// TIA Portal project "hassn_and_musa" (V17)
// Vorlageprojekt für das Buch mit Zielsystem S7-1200

(* hardware
DEVICE "S7-1200-Station_1"  S7-1200 Station
   slot 0: "Baugruppenträger_0"  Rack  V1.0
   slot 1: "PLC_1"  CPU 1211C DC/DC/DC  6ES7 211-1AE40-0XB0  V4.1
DEVICE "HMI_1"  TP700 Comfort
   slot 0: "HMI_1"  TP700 Comfort  6AV2 124-0GC01-0AX0  15.0.0.0
   slot 1: "HMI_RT_1"  TP700 Comfort  6AV2 124-0GC01-0AX0  15.0.0.0
   slot 5: "HMI_1.IE_CP_1"  PROFINET Interface  15.0.0.0
      slot 1: "PROFINET Interface_1"  PROFINET Interface
         slot 1: "Port_1"  Port
         slot 2: "Port_2"  Port
   slot 7: "HMI_1.MPI/DP_CP_1"  MPI/DP Interface  15.0.0.0
*)

// ===== PLC "PLC_1"  CPU 1211C DC/DC/DC =====

VAR_GLOBAL   // PLC tag table "Standard-Variablentabelle"
   "StartButton" AT %I0.0 : Bool;
   "StopButton" AT %I0.1 : Bool;
   "StartLight" AT %Q0.0 : Bool;
   "StopLIght" AT %Q0.1 : Bool;
   "emergency stop" AT %I0.2 : Bool;
   "FlipFlop1" AT %M0.0 : Bool;
   "FlipFlop2" AT %M0.1 : Bool;
   "First Conveyor" AT %Q0.4 : Bool;
   "Second Conveyor" AT %Q0.5 : Bool;
   "Vision Sensor" AT %ID34 : DInt;
   "Third Conveyor" AT %Q0.6 : Bool;
   "pusher" AT %Q0.3 : Bool;
   "pusherbacklimit" AT %I0.3 : Bool;
   "pusherfrontlimit" AT %I0.4 : Bool;
   "SensorForblue" AT %I0.5 : Bool;
   "SensorForGreen" AT %I0.6 : Bool;
   "MoveZBlue" AT %Q0.7 : Bool;
   "MoveZGreen" AT %Q1.0 : Bool;
   "Tag_1" AT %M0.2 : Bool;
   "Tag_2" AT %M0.3 : Bool;
   "Tag_3" AT %M0.4 : Bool;
   "Tag_4" AT %M0.5 : Bool;
   "SensorBlueCount" AT %I0.7 : Bool;
   "SensorGrCount" AT %I1.0 : Bool;
   "Tag_5" AT %M0.6 : Bool;
   "Tag_6" AT %M0.7 : Bool;
   "Tag_7" AT %M1.0 : Bool;
   "Tag_8" AT %M1.1 : Bool;
   "Tag_9" AT %M1.2 : Bool;
END_VAR

DATA_BLOCK "HMI"   // DB1
{ S7_Optimized_Access := 'TRUE' }
VERSION : 0.1
   VAR
      "blue boxes" : Int;
      "Reset Count" : Bool;
      "Green boxes" : Int;
      "emergency hmi" : Bool;
      start : Bool;
      stop : Bool;
   END_VAR
BEGIN
END_DATA_BLOCK

// folder: System blocks/Program resources

DATA_BLOCK "IEC_Counter_0_DB"   // DB2
{ S7_Optimized_Access := 'TRUE' }
AUTHOR : Simatic
FAMILY : IEC
NAME : CNTR
VERSION : 1.0
// stored: InstanceOfName IEC_COUNTER
"IEC_COUNTER"
BEGIN
END_DATA_BLOCK

DATA_BLOCK "IEC_Counter_0_DB_1"   // DB3
{ S7_Optimized_Access := 'TRUE' }
AUTHOR : Simatic
FAMILY : IEC
NAME : CNTR
VERSION : 1.0
// stored: InstanceOfName IEC_COUNTER
"IEC_COUNTER"
BEGIN
END_DATA_BLOCK

// folder: (top level)

FUNCTION "Buttonlights" : Void   // FC1, LAD
{ S7_Optimized_Access := 'TRUE' }
VERSION : 0.1
BEGIN

REGION Network 1
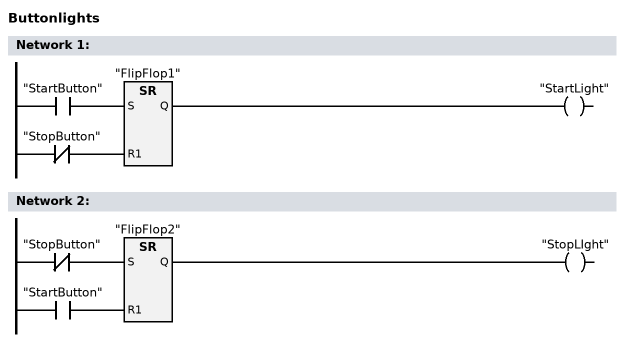
   RUNG wire#powerrail
      Contact( "StartButton" )
      S_SR(operand := "FlipFlop1", r1 := wire#w1)
      Coil( "StartLight" )
   END_RUNG
   RUNG wire#powerrail
      I_Contact( "StopButton" )
   END_RUNG wire#w1
   // the same network as SCL:
   IF "StartButton" THEN
       "FlipFlop1" := TRUE;   // SR flip-flop
   END_IF;
   IF NOT "StopButton" THEN "FlipFlop1" := FALSE; END_IF;
   "StartLight" := "FlipFlop1";
END_REGION

REGION Network 2
   RUNG wire#powerrail
      I_Contact( "StopButton" )
      S_SR(operand := "FlipFlop2", r1 := wire#w1)
      Coil( "StopLIght" )
   END_RUNG
   RUNG wire#powerrail
      Contact( "StartButton" )
   END_RUNG wire#w1
   // the same network as SCL:
   IF NOT "StopButton" THEN
       "FlipFlop2" := TRUE;   // SR flip-flop
   END_IF;
   IF "StartButton" THEN "FlipFlop2" := FALSE; END_IF;
   "StopLIght" := "FlipFlop2";
END_REGION
END_FUNCTION

FUNCTION "StartConvFromFactory" : Void   // FC2, LAD
{ S7_Optimized_Access := 'TRUE' }
VERSION : 0.1
BEGIN

REGION Network 1
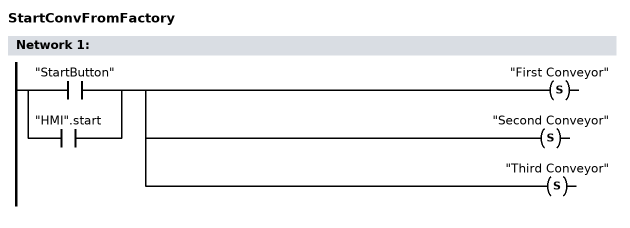
   RUNG wire#powerrail
      Contact( "StartButton" )
      wire#w1
      S_Coil( "First Conveyor" )
   END_RUNG
   RUNG wire#powerrail
      Contact( "HMI".start )
   END_RUNG wire#w1
   RUNG wire#w1
      S_Coil( "Second Conveyor" )
   END_RUNG
   RUNG wire#w1
      S_Coil( "Third Conveyor" )
   END_RUNG
   // the same network as SCL:
   IF "StartButton" OR "HMI".start THEN
       "First Conveyor" := TRUE;
       "Second Conveyor" := TRUE;
       "Third Conveyor" := TRUE;
   END_IF;
END_REGION
END_FUNCTION

FUNCTION "PushGreen" : Void   // FC3, SCL
{ S7_Optimized_Access := 'TRUE' }
VERSION : 0.1
BEGIN

   IF "Vision Sensor" = 4 AND "pusherbacklimit" = 1 THEN
       "pusher" := 1;
   ELSIF "Vision Sensor" <> 4 AND "pusherfrontlimit" = 1 THEN
       "pusher" := 0;
   END_IF;
END_FUNCTION

FUNCTION "Put the tags" : Void   // FC4, LAD
{ S7_Optimized_Access := 'TRUE' }
VERSION : 0.1
   VAR_TEMP   // added for the SCL form of the ladder/FBD networks
      _w1 : Bool;
      _w2 : Bool;
      _w3 : Bool;
      _w4 : Bool;
   END_VAR
BEGIN

REGION Network 1
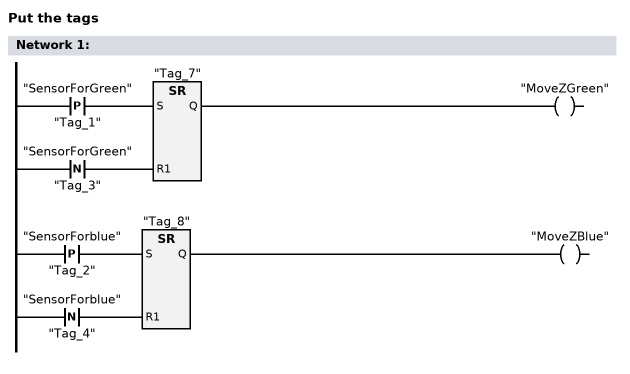
   RUNG wire#powerrail
      P_Contact(operand := "SensorForGreen", bit := "Tag_1")
      S_SR(operand := "Tag_7", r1 := wire#w1)
      Coil( "MoveZGreen" )
   END_RUNG
   RUNG wire#powerrail
      N_Contact(operand := "SensorForGreen", bit := "Tag_3")
   END_RUNG wire#w1
   RUNG wire#powerrail
      P_Contact(operand := "SensorForblue", bit := "Tag_2")
      S_SR(operand := "Tag_8", r1 := wire#w2)
      Coil( "MoveZBlue" )
   END_RUNG
   RUNG wire#powerrail
      N_Contact(operand := "SensorForblue", bit := "Tag_4")
   END_RUNG wire#w2
   // the same network as SCL:
   #_w1 := "SensorForGreen" AND NOT "Tag_1";   // rising edge of "SensorForGreen"
   "Tag_1" := "SensorForGreen";
   #_w2 := NOT "SensorForGreen" AND "Tag_3";   // falling edge of "SensorForGreen"
   "Tag_3" := "SensorForGreen";
   IF #_w1 THEN
       "Tag_7" := TRUE;   // SR flip-flop
   END_IF;
   IF #_w2 THEN "Tag_7" := FALSE; END_IF;
   "MoveZGreen" := "Tag_7";
   #_w3 := "SensorForblue" AND NOT "Tag_2";   // rising edge of "SensorForblue"
   "Tag_2" := "SensorForblue";
   #_w4 := NOT "SensorForblue" AND "Tag_4";   // falling edge of "SensorForblue"
   "Tag_4" := "SensorForblue";
   IF #_w3 THEN
       "Tag_8" := TRUE;   // SR flip-flop
   END_IF;
   IF #_w4 THEN "Tag_8" := FALSE; END_IF;
   "MoveZBlue" := "Tag_8";
END_REGION
END_FUNCTION

FUNCTION "emergency" : Void   // FC5, SCL
{ S7_Optimized_Access := 'TRUE' }
VERSION : 0.1
BEGIN
   WHILE "emergency stop" = 1 OR "HMI"."emergency hmi" = 1 DO
       "SensorForblue" := 0;
       "SensorForGreen" := 0;
       "First Conveyor" := 0;
       "Second Conveyor" := 0;
       "Third Conveyor" := 0;
       "pusher" := 0;
      // "MoveZBlue" := 0;
     //  "MoveZGreen" := 0;
   END_WHILE;
END_FUNCTION

FUNCTION "Count the boxes" : Void   // FC6, LAD
{ S7_Optimized_Access := 'TRUE' }
VERSION : 0.1
   VAR_TEMP   // added for the SCL form of the ladder/FBD networks
      _w1 : Bool;
   END_VAR
BEGIN

REGION Network 1
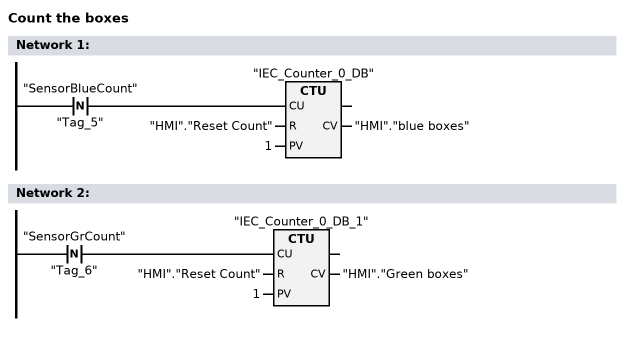
   #_w1 := NOT "SensorBlueCount" AND "Tag_5";   // falling edge of "SensorBlueCount"
   "Tag_5" := "SensorBlueCount";
   "IEC_Counter_0_DB".CTU(CU := #_w1, R := "HMI"."Reset Count", PV := 1, CV => "HMI"."blue boxes");
END_REGION

REGION Network 2
   #_w1 := NOT "SensorGrCount" AND "Tag_6";   // falling edge of "SensorGrCount"
   "Tag_6" := "SensorGrCount";
   "IEC_Counter_0_DB_1".CTU(CU := #_w1, R := "HMI"."Reset Count", PV := 1, CV => "HMI"."Green boxes");
END_REGION
END_FUNCTION

FUNCTION "stop" : Void   // FC7, SCL
{ S7_Optimized_Access := 'TRUE' }
VERSION : 0.1
BEGIN
   //WHILE "StopButton" = 1 DO //OR "HMI".stop = 1 DO
       "SensorForblue" := 0;
       "SensorForGreen" := 0;
       "First Conveyor" := 0;
       "Second Conveyor" := 0;
       "Third Conveyor" := 0;
       "pusher" := 0;
       "MoveZBlue" := 0;
       "MoveZGreen" := 0;
      // END_WHILE;
END_FUNCTION

FUNCTION "MHJ-PLC-Lab-Function-S71200" : Void   // FC9000, SCL
{ S7_Optimized_Access := 'TRUE' }
VERSION : 0.1
   VAR_TEMP
      rdTimeReturn : Int;
      outputTime : DTL;
      SyncVal : Byte;
      forVal : Int;
      forVal_2 : Int;
      Value : Byte;
   END_VAR
   VAR CONSTANT
      CompVal : Byte := 16#34;
      Value_01 : Byte := 16#11;
      Value_01_DW : DWord := 16#A165_D992;
      Value_02_DW : DWord := 16#58BE_4401;
   END_VAR
BEGIN

   #Value:=PEEK(area := 16#82,
        dbNumber := 0,
        byteOffset := 511);
   #Value := #Value + 1;

   POKE(area := 16#82,
        dbNumber := 0,
        byteOffset := 511,
        value := #Value);

   POKE(area:=16#81,
        dbNumber:=0,
        byteOffset:=1016,
        value:=#Value_01_DW);
   POKE(area := 16#81,
        dbNumber := 0,
        byteOffset := 1020,
        value := #Value_02_DW);

   POKE(area := 16#81,
        dbNumber := 0,
        byteOffset := 511,
        value := B#16#00);

   FOR #forVal := 0 TO 120 DO
       FOR #forVal_2:=0 TO 10 DO
           #rdTimeReturn:=RD_SYS_T(#outputTime);
           #rdTimeReturn := WR_SYS_T(#outputTime);
           #rdTimeReturn := RD_SYS_T(#outputTime);
           #rdTimeReturn := WR_SYS_T(#outputTime);
       END_FOR;
       #SyncVal:= PEEK(area := 16#81,
                      dbNumber := 0,
                      byteOffset := 511);
       IF #SyncVal = #CompVal THEN
          GOTO M_1;
       END_IF;
   END_FOR;
   RETURN;

   M_1:
   POKE(area := 16#81,
        dbNumber := 0,
        byteOffset := 511,
        value := B#16#0);
END_FUNCTION

ORGANIZATION_BLOCK "Main"   // OB1, LAD, ProgramCycle
TITLE = "Main Program Sweep (Cycle)"
{ S7_Optimized_Access := 'TRUE' }
VERSION : 0.1
   VAR_INPUT
      Initial_Call : Bool;   // Initial call of this OB
      Remanence : Bool;   // =True, if remanent data are available
   END_VAR
BEGIN

REGION Network 1: Konnektierungsbaustein für PLC-Lab
   // Im Netzwerk 1 wird der Konnektierungsbaustein für PLC-Lab aufgerufen.
   // Dieser Aufruf darf nicht entfernt werden!
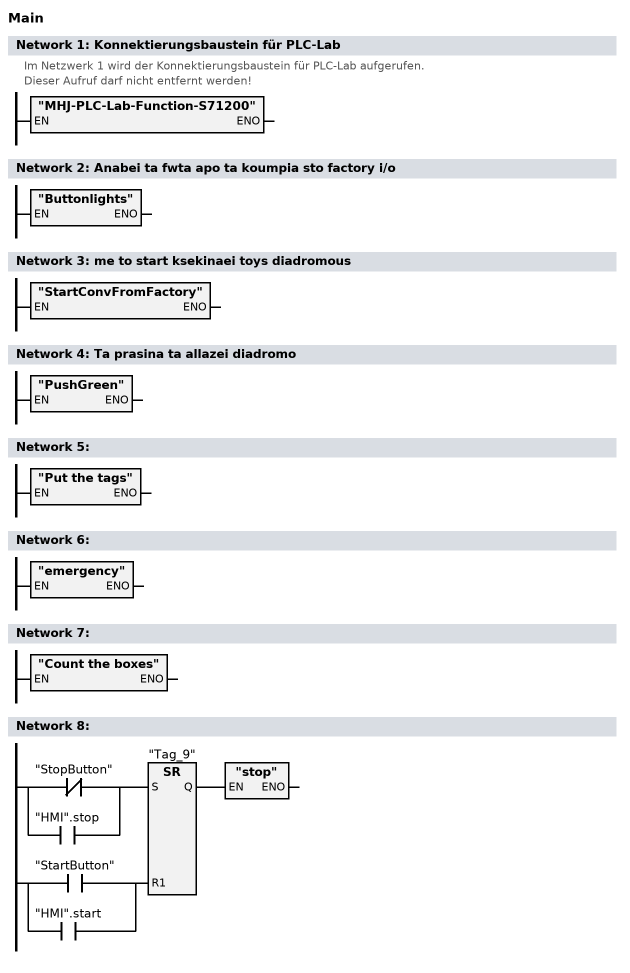
   RUNG wire#powerrail
      "MHJ-PLC-Lab-Function-S71200"()
   END_RUNG
   // the same network as SCL:
   "MHJ-PLC-Lab-Function-S71200"();
END_REGION

REGION Network 2: Anabei ta fwta apo ta koumpia sto factory i/o
   RUNG wire#powerrail
      "Buttonlights"()
   END_RUNG
   // the same network as SCL:
   "Buttonlights"();
END_REGION

REGION Network 3: me to start ksekinaei toys diadromous
   RUNG wire#powerrail
      "StartConvFromFactory"()
   END_RUNG
   // the same network as SCL:
   "StartConvFromFactory"();
END_REGION

REGION Network 4: Ta prasina ta allazei diadromo
   RUNG wire#powerrail
      "PushGreen"()
   END_RUNG
   // the same network as SCL:
   "PushGreen"();
END_REGION

REGION Network 5
   RUNG wire#powerrail
      "Put the tags"()
   END_RUNG
   // the same network as SCL:
   "Put the tags"();
END_REGION

REGION Network 6
   RUNG wire#powerrail
      "emergency"()
   END_RUNG
   // the same network as SCL:
   "emergency"();
END_REGION

REGION Network 7
   RUNG wire#powerrail
      "Count the boxes"()
   END_RUNG
   // the same network as SCL:
   "Count the boxes"();
END_REGION

REGION Network 8
   RUNG wire#powerrail
      I_Contact( "StopButton" )
      wire#w1
      S_SR(operand := "Tag_9", r1 := wire#w2)
      "stop"()
   END_RUNG
   RUNG wire#powerrail
      Contact( "HMI".stop )
   END_RUNG wire#w1
   RUNG wire#powerrail
      Contact( "StartButton" )
   END_RUNG wire#w2
   RUNG wire#powerrail
      Contact( "HMI".start )
   END_RUNG wire#w2
   // the same network as SCL:
   IF NOT "StopButton" OR "HMI".stop THEN
       "Tag_9" := TRUE;   // SR flip-flop
   END_IF;
   IF "StartButton" OR "HMI".start THEN "Tag_9" := FALSE; END_IF;
   IF "Tag_9" THEN "stop"(); END_IF;
END_REGION
END_ORGANIZATION_BLOCK

(* ===== HMI "HMI_RT_1" =====
system functions are stored by id; their names below are inferred from use
connection "HMI_Connection_1": ETHERNET, S7_1200_OMS

HMI tags "Default tag table"
   "Tag_ScreenNumber" : UInt, internal
   "HMI_blue boxes" : Int = PLC HMI."blue boxes", 1 s
   "HMI_Green boxes" : Int = PLC HMI."Green boxes", 1 s
   "emergency stop" : Bool = PLC "emergency stop" AT %I0.2, 1 s
   "HMI_Reset Count" : Bool = PLC HMI."Reset Count", 1 s
   "HMI_emergency hmi" : Bool = PLC HMI."emergency hmi", 1 s
   "StartButton" : Bool = PLC StartButton AT %I0.0, 1 s
   "StopButton" : Bool = PLC StopButton AT %I0.1, 1 s
   "HMI_start" : Bool = PLC HMI.start, 1 s
   "HMI_stop" : Bool = PLC HMI.stop, 1 s

screen "Root screen" 800x420, template "Template_1"
   on GenerateScreen: SetTag("Tag_ScreenNumber", 1)
   TextField "Text field_1" at 218,106 size 16x23; Text 'Text'
   IOField "I/O field_1" at 126,228 size 96x32; FormatPattern 99999
      ProcessValue <- "HMI_blue boxes"
   IOField "I/O field_2" at 126,267 size 96x32; FormatPattern 99999
      ProcessValue <- "HMI_Green boxes"
   TextField "Text field_2" at 14,233 size 112x23; Text 'Blue Boxes:'
   TextField "Text field_3" at 14,272 size 112x23; Text 'Blue Boxes:'
   Button "Button_1" at 14,170 size 133x42; TextOff 'Reset Counters'
      on Press: function_b14e0dd5("HMI_Reset Count", 0)
   Button "Button_2" at 13,13 size 133x42; TextOff 'Start'
      on Press: function_b14e0dd5("HMI_start", 0)
   Button "Button_3" at 13,72 size 133x42; TextOff 'Stop'
      on Press: function_b14e0dd5("HMI_stop", 0)
   Switch "Switch_1" at 288,0 size 240x61; CaptionText 'EMERGENCY STOP'; TextOff 'OFF'; TextOn 'ON'
      ProcessValue <- "HMI_emergency hmi"

Template "Template_1" 800x420
   Button "Exit" at 720,360 size 78x58; TextOff 'Exit'; PictureOff "ExitRuntime_TP700_Comfort_TR"; PictureOn "ExitRuntime_TP700_Comfort_TR"
      on Release: StopRuntime(0)
   Button "Template_Button" at 640,360 size 78x58; TextOff 'Text'
   Button "Template_Button_1" at 560,360 size 78x58; TextOff 'Text'
   Button "Template_Button_2" at 480,360 size 78x58; TextOff 'Text'
   Button "Template_Button_3" at 400,360 size 78x58; TextOff 'Text'
   Button "Template_Button_4" at 321,360 size 78x58; TextOff 'Text'
   Button "Template_Button_5" at 241,360 size 78x58; TextOff 'Text'
   Button "Template_Button_6" at 161,360 size 78x58; TextOff 'Text'
   Button "Alarms" at 81,360 size 78x58; TextOff 'Alarms'; PictureOff "AlarmDisplay_TP700_Comfort_TR"; PictureOn "AlarmDisplay_TP700_Comfort_TR"
      on Release: function_ef3f5d25("Alarm window_Unacknowledged", -1)
   Button "Start screen" at 1,360 size 78x58; TextOff 'Start screen'; PictureOff "NavigateHome_TP700_Comfort_TR"; PictureOn "NavigateHome_TP700_Comfort_TR"
      on Release: ActivateScreen("Root screen", 0)
*)